PROGRAM pump_control
VAR
	//Repeat for each pump?
	pump_1_enable: BOOL;
	pump_1_auto_request: BOOL;
	pump_1_cip_request: BOOL;
	pump_1_manual_request: BOOL;
	pump_1_stop_request: BOOL;
	pump_1_intlk: BOOL;
	gen_alm_active: BOOL;
	ed_routine_auto: BOOL;
	ed_routine_cip: BOOL;
	ed_routine_manual: BOOL;
END_VAR

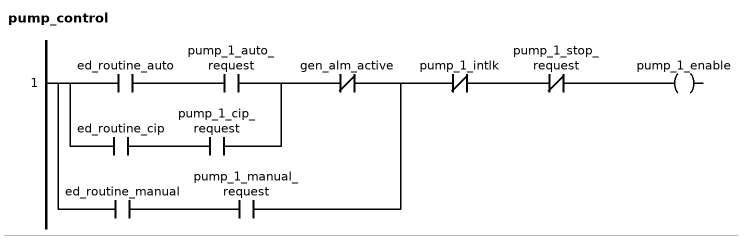
// NETWORK 1
pump_1_enable := ((ed_routine_auto AND pump_1_auto_request OR ed_routine_cip AND pump_1_cip_request) AND NOT gen_alm_active OR ed_routine_manual AND pump_1_manual_request) AND NOT pump_1_intlk AND NOT pump_1_stop_request;

END_PROGRAM

(* stored: Version 1.1.0.1, ProductVersion 3.1.4024.12
   POU pump_control: Id {3b5ad67c-a464-4c74-9317-fc4708b2e954}, SpecialFunc None *)
